# B&R Automation Studio project laba1
Automation Studio 4.5.2.102

## Configuration laba1

### Hardware
```
4PP065_0571_P74 : 4PP065.0571-P74 v1.2.0.0
  Connector IF5:
    ActivateDevice = 1
    Mode = Manual
    InternetAddress = 10.0.1.10
    SubnetMask = 255.255.255.0
  ConfigurationID = labBR
  Simulation = 1
```

## Logical view

### Library Logical/Libraries/Library

#### Library.fun
```iecst
{REDUND_ERROR} {REDUND_UNREPLICABLE} FUNCTION_BLOCK FB_Integrator (*TODO: Add your comment here*) (*$GROUP=User,$CAT=User,$GROUPICON=User.png,$CATICON=User.png*)
	VAR_INPUT
		in : {REDUND_UNREPLICABLE} REAL;
	END_VAR
	VAR_OUTPUT
		out : {REDUND_UNREPLICABLE} REAL;
	END_VAR
	VAR
		dt : {REDUND_UNREPLICABLE} REAL;
		prev_value : {REDUND_UNREPLICABLE} REAL;
	END_VAR
END_FUNCTION_BLOCK

{REDUND_ERROR} {REDUND_UNREPLICABLE} FUNCTION_BLOCK FB_Motor (*TODO: Add your comment here*) (*$GROUP=User,$CAT=User,$GROUPICON=User.png,$CATICON=User.png*)
	VAR_INPUT
		u : {REDUND_UNREPLICABLE} REAL;
	END_VAR
	VAR_OUTPUT
		w : {REDUND_UNREPLICABLE} REAL;
		phi : {REDUND_UNREPLICABLE} REAL;
	END_VAR
	VAR
		integrator : {REDUND_UNREPLICABLE} FB_Integrator;
		Tm : {REDUND_UNREPLICABLE} REAL;
		ke : {REDUND_UNREPLICABLE} REAL;
		dt : {REDUND_UNREPLICABLE} REAL;
		prev_w : {REDUND_UNREPLICABLE} REAL;
		prev_phi : {REDUND_UNREPLICABLE} REAL;
	END_VAR
END_FUNCTION_BLOCK

{REDUND_ERROR} {REDUND_UNREPLICABLE} FUNCTION_BLOCK FB_Regulator (*TODO: Add your comment here*) (*$GROUP=User,$CAT=User,$GROUPICON=User.png,$CATICON=User.png*)
	VAR_INPUT
		e : {REDUND_UNREPLICABLE} REAL;
	END_VAR
	VAR_OUTPUT
		u : {REDUND_UNREPLICABLE} REAL;
	END_VAR
	VAR
		k_p : {REDUND_UNREPLICABLE} REAL;
		k_i : {REDUND_UNREPLICABLE} REAL;
		integrator : {REDUND_UNREPLICABLE} FB_Integrator;
		iyOld : {REDUND_UNREPLICABLE} REAL;
		max_abs_value : {REDUND_UNREPLICABLE} REAL;
		dt : {REDUND_UNREPLICABLE} REAL;
		prev_value : {REDUND_UNREPLICABLE} REAL;
		temp : {REDUND_UNREPLICABLE} REAL;
	END_VAR
END_FUNCTION_BLOCK
```

#### FB_Integrator.c
```c
#include <bur/plctypes.h>
#ifdef __cplusplus
	extern "C"
	{
#endif
	#include "Library.h"
#ifdef __cplusplus
	};
#endif
/* TODO: Add your comment here */
void FB_Integrator(struct FB_Integrator* inst)
{
	inst->dt = 0.01;
	inst->out = inst->dt*inst->in + inst->prev_value;
	inst->prev_value = inst->out;
}
```

#### FB_Motor.c
```c
#include <bur/plctypes.h>
#ifdef __cplusplus
	extern "C"
	{
#endif
	#include "Library.h"
#ifdef __cplusplus
	};
#endif
/* TODO: Add your comment here */
void FB_Motor(struct FB_Motor* inst)
{
	inst->dt = 0.01;

	inst->integrator.in = ((inst->u / inst->ke) - inst->w) / inst->Tm;
	FB_Integrator(&inst->integrator);
	inst->w = inst->integrator.out;

}
```

#### FB_Regulator.c
```c
#include <bur/plctypes.h>
#ifdef __cplusplus
	extern "C"
	{
#endif
	#include "Library.h"
#ifdef __cplusplus
	};
#endif
/* TODO: Add your comment here */
/*void FB_Regulator(struct FB_Regulator* inst)
{
	inst->dt = 0.01;
	inst->integrator.in = (inst->e * inst->k_i) + inst->iyOld;
	FB_Integrator(&inst->integrator);
	if (abs(inst->e * inst->k_p) > inst->max_abs_value)
	{
		if (abs(inst->max_abs_value + inst->integrator.out) > inst->max_abs_value)
		{
			inst->u = inst->max_abs_value;
			inst->iyOld = inst->max_abs_value;
		}
		else
		{
			inst->u = inst->max_abs_value + inst->integrator.out;
			inst->iyOld = 0;
		}
	}
	else
	{
		if (abs((inst->e * inst->k_p) + inst->integrator.out) > inst->max_abs_value)
		{
			inst->u = inst->max_abs_value;
			inst->iyOld = inst->max_abs_value - (inst->e * inst->k_p);
		}
		else
		{
			inst->u = (inst->e * inst->k_p) + inst->integrator.out;
			inst->iyOld = 0;
		}
	}
} */

void FB_Regulator(struct FB_Regulator* inst)
{
	REAL a = inst ->e * inst -> k_p;
	REAL b = inst ->e * inst -> k_i;

	a = a > inst -> max_abs_value ? inst ->max_abs_value : a;
	a = a < -inst -> max_abs_value ? -inst ->max_abs_value : a;

	inst -> integrator.in = b + inst -> iyOld;
	FB_Integrator (&inst -> integrator);

	REAL sum = a + inst -> integrator.out;

	inst -> u = sum;
	inst -> u = inst -> u > inst -> max_abs_value ? inst -> max_abs_value : inst -> u;
	inst -> u = inst -> u < -inst -> max_abs_value ? -inst -> max_abs_value : inst -> u;

	inst -> iyOld = inst ->u - sum;
}
```

### Program Logical/Program

#### Variables.var
```iecst
VAR
	fb_motor1 : {REDUND_UNREPLICABLE} FB_Motor;
	fb_motor2 : {REDUND_UNREPLICABLE} FB_Motor;
	fb_regulator : {REDUND_UNREPLICABLE} FB_Regulator;
	Speed : {REDUND_UNREPLICABLE} REAL;
	Enable : {REDUND_UNREPLICABLE} BOOL;
	counter : {REDUND_UNREPLICABLE} UINT;
END_VAR
```

#### Cyclic.c
```c
#include <bur/plctypes.h>

#ifdef _DEFAULT_INCLUDES
	#include <AsDefault.h>
#endif

void _CYCLIC ProgramCyclic(void)
{
	if (Enable)
	{
		if (counter == 200)
		{
			Speed = 0;
			counter = 0;
		}
		if (counter == 50)
		{
			Speed = 50;
		}

		counter++;

		fb_regulator.e = Speed - fb_motor1.w;
		FB_Regulator(&fb_regulator);
		fb_motor1.u = fb_regulator.u;

		FB_Motor(&fb_motor1);

		fb_motor2.u = Speed * fb_motor2.ke;
		FB_Motor(&fb_motor2);
		}

}
```

#### Init.c
```c
#include <bur/plctypes.h>

#ifdef _DEFAULT_INCLUDES
	#include <AsDefault.h>
#endif

void _INIT ProgramInit(void)
{
	fb_motor1.dt = 0.01;
	fb_motor1.ke = 0.0011;
	fb_motor1.Tm = 0.0246;
	fb_motor1.u = 60;
	fb_motor1.integrator.dt = 0.01;

	fb_motor2.dt = 0.01;
	fb_motor2.ke = 0.0011;
	fb_motor2.Tm = 0.0246;
	fb_motor2.u = 0;
	fb_motor2.integrator.dt = 0.01;

	fb_regulator.dt = 0.01;
	fb_regulator.integrator.dt = 0.01;
	fb_regulator.k_p = 0.0006;
	fb_regulator.k_i = 0.0228;
	fb_regulator.max_abs_value = 24.0;

	Speed = 0;
	counter = 0;

}
```
